FUNCTION_BLOCK MUL_SINT (* IEC 61131-3 SINT Multiplication *)
  (* Standard: 61131-3 *)
  (* Version 0.0, 2004-12-15, JHC, Rockwell Automation, Converted from SRC format. *)
  (* Compiler header: package fb.rt.plc.math; *)
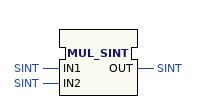
  VAR_INPUT
    IN1 : SINT; (* Multiplicand *)
    IN2 : SINT; (* Multiplier *)
  END_VAR
  VAR_OUTPUT
    OUT : SINT; (* Product *)
  END_VAR
END_FUNCTION_BLOCK
